stInitData.ModelParameters._R[9672] := 0.3081594558900842;
stInitData.ModelParameters._R[9673] := 0.49119037988082304;
stInitData.ModelParameters._R[9674] := 0.54802588103738414;
stInitData.ModelParameters._R[9675] := 0.5766695935703896;
stInitData.ModelParameters._R[9676] := 0.90517499100223242;
stInitData.ModelParameters._R[9677] := 0.32631200684456385;
stInitData.ModelParameters._R[9678] := 0.31554996521816614;
stInitData.ModelParameters._R[9679] := 0.58613432693044454;
stInitData.ModelParameters._R[9680] := 0.98725103325684738;
stInitData.ModelParameters._R[9681] := 0.39443656608666267;
stInitData.ModelParameters._R[9682] := 0.52590831780389014;
stInitData.ModelParameters._R[9683] := 0.33277164828551653;
stInitData.ModelParameters._R[9684] := 0.57697613821259108;
stInitData.ModelParameters._R[9685] := 0.59470626591824982;
stInitData.ModelParameters._R[9686] := 0.97728509593354573;
stInitData.ModelParameters._R[9687] := 0.6473974259604981;
stInitData.ModelParameters._R[9688] := 0.58921948813149061;
stInitData.ModelParameters._R[9689] := 0.77679355501374725;
stInitData.ModelParameters._R[9690] := 0.79979586848841022;
stInitData.ModelParameters._R[9691] := 0.20195251741029296;
stInitData.ModelParameters._R[9692] := 0.85091439584456219;
stInitData.ModelParameters._R[9693] := 0.27732676922075522;
stInitData.ModelParameters._R[9694] := 0.13292198388144139;
stInitData.ModelParameters._R[9695] := 0.27889231958345484;
stInitData.ModelParameters._R[9696] := 0.13763582277844255;
stInitData.ModelParameters._R[9697] := 0.33151232005878017;
stInitData.ModelParameters._R[9698] := 0.35145746439539727;
stInitData.ModelParameters._R[9699] := 0.36038726014308942;
stInitData.ModelParameters._R[9700] := 0.88193994244801943;
stInitData.ModelParameters._R[9701] := 0.9328112379804081;
stInitData.ModelParameters._R[9702] := 0.52121737425116754;
stInitData.ModelParameters._R[9703] := 0.7103941054557622;
stInitData.ModelParameters._R[9704] := 0.35591153481502213;
stInitData.ModelParameters._R[9705] := 0.30623573374135654;
stInitData.ModelParameters._R[9706] := 0.32448345869195733;
stInitData.ModelParameters._R[9707] := 0.25705792007434003;
stInitData.ModelParameters._R[9708] := 0.3001442867159051;
stInitData.ModelParameters._R[9709] := 0.71709970026557601;
stInitData.ModelParameters._R[9710] := 0.30537705430913215;
stInitData.ModelParameters._R[9711] := 0.40321743117402664;
stInitData.ModelParameters._R[9712] := 0.27289617464252264;
stInitData.ModelParameters._R[9713] := 0.57746419995378429;
stInitData.ModelParameters._R[9714] := 0.26762305834442551;
stInitData.ModelParameters._R[9715] := 0.2079714576941572;
stInitData.ModelParameters._R[9716] := 0.61443612128773306;
stInitData.ModelParameters._R[9717] := 0.14638196023715569;
stInitData.ModelParameters._R[9718] := 0.31171678328575386;
stInitData.ModelParameters._R[9719] := 0.17149049807118483;
stInitData.ModelParameters._R[9720] := 0.57987505218000635;
stInitData.ModelParameters._R[9721] := 0.59377132590735826;
stInitData.ModelParameters._R[9722] := 0.6228873515215011;
stInitData.ModelParameters._R[9723] := 0.35302883122952955;
stInitData.ModelParameters._R[9724] := 0.40866668302305986;
stInitData.ModelParameters._R[9725] := 0.39587181913887326;
stInitData.ModelParameters._R[9726] := 0.54428758424609014;
stInitData.ModelParameters._R[9727] := 0.74730280479554523;
stInitData.ModelParameters._R[9728] := 0.94126198539625039;
stInitData.ModelParameters._R[9729] := 0.75262284046442718;
stInitData.ModelParameters._R[9730] := 0.86419193265417726;
stInitData.ModelParameters._R[9731] := 0.97527451192212322;
stInitData.ModelParameters._R[9732] := 0.29691036623971701;
stInitData.ModelParameters._R[9733] := 0.3068750345184541;
stInitData.ModelParameters._R[9734] := 0.77801117617079574;
stInitData.ModelParameters._R[9735] := 0.52013899813102715;
stInitData.ModelParameters._R[9736] := 0.2159352389037883;
stInitData.ModelParameters._R[9737] := 0.48481560477638852;
stInitData.ModelParameters._R[9738] := 0.12702521089252394;
stInitData.ModelParameters._R[9739] := 0.23393696455088481;
stInitData.ModelParameters._R[9740] := 0.48627931050982687;
stInitData.ModelParameters._R[9741] := 0.78567517414504673;
stInitData.ModelParameters._R[9742] := 0.54289188771994268;
stInitData.ModelParameters._R[9743] := 0.35461820603697103;
stInitData.ModelParameters._R[9744] := 0.74780959726572205;
stInitData.ModelParameters._R[9745] := 0.67060317596121843;
stInitData.ModelParameters._R[9746] := 0.36062560169371338;
stInitData.ModelParameters._R[9747] := 0.76906602867914209;
stInitData.ModelParameters._R[9748] := 0.22247379637105591;
stInitData.ModelParameters._R[9749] := 0.96905625932380479;
stInitData.ModelParameters._R[9750] := 0.40699850966949458;
stInitData.ModelParameters._R[9751] := 0.79115939448714923;
stInitData.ModelParameters._R[9752] := 0.16890137358512397;
stInitData.ModelParameters._R[9753] := 0.42572836100797307;
stInitData.ModelParameters._R[9754] := 0.77986861062425639;
stInitData.ModelParameters._R[9755] := 0.96207793323773094;
stInitData.ModelParameters._R[9756] := 0.22836627769795068;
stInitData.ModelParameters._R[9757] := 0.36656334684361447;
stInitData.ModelParameters._R[9758] := 0.50011212685405437;
stInitData.ModelParameters._R[9759] := 0.10456968130595451;
stInitData.ModelParameters._R[9760] := 0.15291139386198394;
stInitData.ModelParameters._R[9761] := 0.72974999584542732;
stInitData.ModelParameters._R[9762] := 0.65151577378750392;
stInitData.ModelParameters._R[9763] := 0.72156165708286868;
stInitData.ModelParameters._R[9764] := 0.80533056043207263;
stInitData.ModelParameters._R[9765] := 0.3297540892709695;
stInitData.ModelParameters._R[9766] := 0.60249604863206108;
stInitData.ModelParameters._R[9767] := 0.29782552474488438;
stInitData.ModelParameters._R[9768] := 0.46509663904829945;
stInitData.ModelParameters._R[9769] := 0.83428493040856078;
stInitData.ModelParameters._R[9770] := 0.71249641952461906;
stInitData.ModelParameters._R[9771] := 0.30706070288783721;
stInitData.ModelParameters._R[9772] := 0.38961451708477912;
stInitData.ModelParameters._R[9773] := 0.28134385898356995;
stInitData.ModelParameters._R[9774] := 0.89810290091873457;
stInitData.ModelParameters._R[9775] := 0.62599877661269654;
stInitData.ModelParameters._R[9776] := 0.68892576012802009;
stInitData.ModelParameters._R[9777] := 0.35704014267279738;
stInitData.ModelParameters._R[9778] := 0.68552692558681905;
stInitData.ModelParameters._R[9779] := 0.46506801392177066;
stInitData.ModelParameters._R[9780] := 0.44827602984733361;
stInitData.ModelParameters._R[9781] := 0.60117405420418724;
stInitData.ModelParameters._R[9782] := 0.8598356559692204;
stInitData.ModelParameters._R[9783] := 0.14471334839153888;
stInitData.ModelParameters._R[9784] := 0.43374441264226504;
stInitData.ModelParameters._R[9785] := 0.83259316843209541;
stInitData.ModelParameters._R[9786] := 0.77691378154641844;
stInitData.ModelParameters._R[9787] := 0.41185978879895524;
stInitData.ModelParameters._R[9788] := 0.86809696188712371;
stInitData.ModelParameters._R[9789] := 0.45202449896875896;
stInitData.ModelParameters._R[9790] := 0.47387995480326295;
stInitData.ModelParameters._R[9791] := 0.37373938212944169;
stInitData.ModelParameters._R[9792] := 0.47203881799654901;
stInitData.ModelParameters._R[9793] := 0.21665736950560788;
stInitData.ModelParameters._R[9794] := 0.71193845643467191;
stInitData.ModelParameters._R[9795] := 0.60087178778721784;
stInitData.ModelParameters._R[9796] := 0.18480381185150935;
stInitData.ModelParameters._R[9797] := 0.61156038279243841;
stInitData.ModelParameters._R[9798] := 0.48881534640862712;
stInitData.ModelParameters._R[9799] := 0.2887492582190212;
stInitData.ModelParameters._R[9800] := 0.90560748438258731;
stInitData.ModelParameters._R[9801] := 0.91282438528684806;
stInitData.ModelParameters._R[9802] := 0.93933814790319115;
stInitData.ModelParameters._R[9803] := 0.46333753107322218;
stInitData.ModelParameters._R[9804] := 0.50569000162206179;
stInitData.ModelParameters._R[9805] := 0.30566404573220807;
stInitData.ModelParameters._R[9806] := 0.64965225594956377;
stInitData.ModelParameters._R[9807] := 0.70292342688034215;
stInitData.ModelParameters._R[9808] := 0.13905092695678048;
stInitData.ModelParameters._R[9809] := 0.97994981053390018;
stInitData.ModelParameters._R[9810] := 0.43445130700397561;
stInitData.ModelParameters._R[9811] := 0.31506443138868001;
stInitData.ModelParameters._R[9812] := 0.85757506749587809;
stInitData.ModelParameters._R[9813] := 0.1763294640582358;
stInitData.ModelParameters._R[9814] := 0.69769559239292012;
stInitData.ModelParameters._R[9815] := 0.98351187446968924;
stInitData.ModelParameters._R[9816] := 0.98809332311749754;
stInitData.ModelParameters._R[9817] := 0.24972506295303096;
stInitData.ModelParameters._R[9818] := 0.29677807389335964;
stInitData.ModelParameters._R[9819] := 0.7310455966023609;
stInitData.ModelParameters._R[9820] := 0.70509892202199953;
stInitData.ModelParameters._R[9821] := 0.86081634813716212;
stInitData.ModelParameters._R[9822] := 0.18440328527322083;
stInitData.ModelParameters._R[9823] := 0.79295740209692889;
stInitData.ModelParameters._R[9824] := 0.21655927614605064;
stInitData.ModelParameters._R[9825] := 0.81458404577631305;
stInitData.ModelParameters._R[9826] := 0.91417569866210047;
stInitData.ModelParameters._R[9827] := 0.53598273335743885;
stInitData.ModelParameters._R[9828] := 0.13001393050244439;
stInitData.ModelParameters._R[9829] := 0.42674438764497558;
stInitData.ModelParameters._R[9830] := 0.43386560348008019;
stInitData.ModelParameters._R[9831] := 0.92167093241993181;
stInitData.ModelParameters._R[9832] := 0.53657613107005286;
stInitData.ModelParameters._R[9833] := 0.47039575501314101;
stInitData.ModelParameters._R[9834] := 0.12185679425336628;
stInitData.ModelParameters._R[9835] := 0.69983295137423684;
stInitData.ModelParameters._R[9836] := 0.33035427524428851;
stInitData.ModelParameters._R[9837] := 0.95589594052270166;
stInitData.ModelParameters._R[9838] := 0.88544502057114216;
stInitData.ModelParameters._R[9839] := 0.21414976605871799;
stInitData.ModelParameters._R[9840] := 0.3238939102341406;
stInitData.ModelParameters._R[9841] := 0.77378392527788453;
stInitData.ModelParameters._R[9842] := 0.96786698139501082;
stInitData.ModelParameters._R[9843] := 0.11756317333129397;
stInitData.ModelParameters._R[9844] := 0.81129960834296344;
stInitData.ModelParameters._R[9845] := 0.11523464413150972;
stInitData.ModelParameters._R[9846] := 0.21190597514665205;
stInitData.ModelParameters._R[9847] := 0.25786608897761082;
stInitData.ModelParameters._R[9848] := 0.58976475816634866;
stInitData.ModelParameters._R[9849] := 0.18870306172612777;
stInitData.ModelParameters._R[9850] := 0.24374627352027151;
stInitData.ModelParameters._R[9851] := 0.59687413219332952;
stInitData.ModelParameters._R[9852] := 0.88938063303810577;
stInitData.ModelParameters._R[9853] := 0.48799895426478723;
stInitData.ModelParameters._R[9854] := 0.66841219131362539;
stInitData.ModelParameters._R[9855] := 0.36963265944559598;
stInitData.ModelParameters._R[9856] := 0.82943424578666913;
stInitData.ModelParameters._R[9857] := 0.52837834484509139;
stInitData.ModelParameters._R[9858] := 0.78124555273882812;
stInitData.ModelParameters._R[9859] := 0.89411646635390996;
stInitData.ModelParameters._R[9860] := 0.44655796563814998;
stInitData.ModelParameters._R[9861] := 0.26907291506530817;
stInitData.ModelParameters._R[9862] := 0.90306949756615351;
stInitData.ModelParameters._R[9863] := 0.49719892918312592;
stInitData.ModelParameters._R[9864] := 0.39060635402980037;
stInitData.ModelParameters._R[9865] := 0.56296943485308804;
stInitData.ModelParameters._R[9866] := 0.60029370508560109;
stInitData.ModelParameters._R[9867] := 0.20633785991571885;
stInitData.ModelParameters._R[9868] := 0.75394922437920553;
stInitData.ModelParameters._R[9869] := 0.51501421427446903;
stInitData.ModelParameters._R[9870] := 0.6656375285467182;
stInitData.ModelParameters._R[9871] := 0.8977548300710646;
stInitData.ModelParameters._R[9872] := 0.68278844051304932;
stInitData.ModelParameters._R[9873] := 0.61816206649149363;
stInitData.ModelParameters._R[9874] := 0.91143009974599742;
stInitData.ModelParameters._R[9875] := 0.94326207364445436;
stInitData.ModelParameters._R[9876] := 0.5115350512905229;
stInitData.ModelParameters._R[9877] := 0.24682020951989475;
stInitData.ModelParameters._R[9878] := 0.18152125255983564;
stInitData.ModelParameters._R[9879] := 0.77840909392712043;
stInitData.ModelParameters._R[9880] := 0.383904375066493;
stInitData.ModelParameters._R[9881] := 0.21915716447704253;
stInitData.ModelParameters._R[9882] := 0.56995532127121473;
stInitData.ModelParameters._R[9883] := 0.40433296362694537;
stInitData.ModelParameters._R[9884] := 0.11836991444730471;
stInitData.ModelParameters._R[9885] := 0.90923916899573165;
stInitData.ModelParameters._R[9886] := 0.58802008711548659;
stInitData.ModelParameters._R[9887] := 0.75842061053208376;
stInitData.ModelParameters._R[9888] := 0.65446898207421211;
stInitData.ModelParameters._R[9889] := 0.32221721211912274;
stInitData.ModelParameters._R[9890] := 0.48455431451698294;
stInitData.ModelParameters._R[9891] := 0.22037638529936665;
stInitData.ModelParameters._R[9892] := 0.24955994595845665;
stInitData.ModelParameters._R[9893] := 0.6046791376096643;
stInitData.ModelParameters._R[9894] := 0.34097230707455695;
stInitData.ModelParameters._R[9895] := 0.26855284583115951;
stInitData.ModelParameters._R[9896] := 0.82031413680043519;
stInitData.ModelParameters._R[9897] := 0.89125135895419438;
stInitData.ModelParameters._R[9898] := 0.76446758389946656;
stInitData.ModelParameters._R[9899] := 0.52695820601449106;
stInitData.ModelParameters._R[9900] := 0.27559007504240551;
stInitData.ModelParameters._R[9901] := 0.10212010932597458;
stInitData.ModelParameters._R[9902] := 0.1242068193691995;
stInitData.ModelParameters._R[9903] := 0.37788681109071742;
stInitData.ModelParameters._R[9904] := 0.83272941043909587;
stInitData.ModelParameters._R[9905] := 0.26340634971484178;
stInitData.ModelParameters._R[9906] := 0.18218572649490977;
stInitData.ModelParameters._R[9907] := 0.32245904283530485;
stInitData.ModelParameters._R[9908] := 0.86568668088888945;
stInitData.ModelParameters._R[9909] := 0.13974802192888491;
stInitData.ModelParameters._R[9910] := 0.59516193834479858;
stInitData.ModelParameters._R[9911] := 0.76483707879202056;
stInitData.ModelParameters._R[9912] := 0.51143841182357086;
stInitData.ModelParameters._R[9913] := 0.39162845679447655;
stInitData.ModelParameters._R[9914] := 0.53876455011802438;
stInitData.ModelParameters._R[9915] := 0.45695097931081197;
stInitData.ModelParameters._R[9916] := 0.24462842999048356;
stInitData.ModelParameters._R[9917] := 0.53046316360152046;
stInitData.ModelParameters._R[9918] := 0.54925684421213938;
stInitData.ModelParameters._R[9919] := 0.51839003720238519;
stInitData.ModelParameters._R[9920] := 0.97064456541005695;
stInitData.ModelParameters._R[9921] := 0.5085792426367588;
stInitData.ModelParameters._R[9922] := 0.25989320732517956;
stInitData.ModelParameters._R[9923] := 0.67273895419636554;
stInitData.ModelParameters._R[9924] := 0.43178574153741212;
stInitData.ModelParameters._R[9925] := 0.67761621816188444;
stInitData.ModelParameters._R[9926] := 0.89537055173038982;
stInitData.ModelParameters._R[9927] := 0.37394490472178032;
stInitData.ModelParameters._R[9928] := 0.42633607011448826;
stInitData.ModelParameters._R[9929] := 0.95461521398069504;
stInitData.ModelParameters._R[9930] := 0.12157880126117859;
stInitData.ModelParameters._R[9931] := 0.34322859860874877;
stInitData.ModelParameters._R[9932] := 0.67040877835156609;
stInitData.ModelParameters._R[9933] := 0.50805909243936709;
stInitData.ModelParameters._R[9934] := 0.33646038691757413;
stInitData.ModelParameters._R[9935] := 0.50487648159022047;
stInitData.ModelParameters._R[9936] := 0.48474990849157351;
stInitData.ModelParameters._R[9937] := 0.83218824319015583;
stInitData.ModelParameters._R[9938] := 0.58104809770634869;
stInitData.ModelParameters._R[9939] := 0.99475295605039737;
stInitData.ModelParameters._R[9940] := 0.96769216848124218;
stInitData.ModelParameters._R[9941] := 0.98801487477731365;
stInitData.ModelParameters._R[9942] := 0.60904945047017345;
stInitData.ModelParameters._R[9943] := 0.2646022736436987;
stInitData.ModelParameters._R[9944] := 0.7414170990710871;
stInitData.ModelParameters._R[9945] := 0.731903915379436;
stInitData.ModelParameters._R[9946] := 0.32519407164893999;
stInitData.ModelParameters._R[9947] := 0.87587235810615294;
stInitData.ModelParameters._R[9948] := 0.19665848717129264;
stInitData.ModelParameters._R[9949] := 0.10971892485465168;
stInitData.ModelParameters._R[9950] := 0.50439342672529575;
stInitData.ModelParameters._R[9951] := 0.22104375737750892;
stInitData.ModelParameters._R[9952] := 0.70265879009455434;
stInitData.ModelParameters._R[9953] := 0.95769300417984582;
stInitData.ModelParameters._R[9954] := 0.90474959849072878;
stInitData.ModelParameters._R[9955] := 0.68454510827887072;
stInitData.ModelParameters._R[9956] := 0.37560133540865548;
stInitData.ModelParameters._R[9957] := 0.77528505338122833;
stInitData.ModelParameters._R[9958] := 0.89090794989770672;
stInitData.ModelParameters._R[9959] := 0.33569319079658316;
stInitData.ModelParameters._R[9960] := 0.57809660926134632;
stInitData.ModelParameters._R[9961] := 0.44644731935988691;
stInitData.ModelParameters._R[9962] := 0.66518006373582306;
stInitData.ModelParameters._R[9963] := 0.11587791613012297;
stInitData.ModelParameters._R[9964] := 0.66962135407134016;
stInitData.ModelParameters._R[9965] := 0.65411366157139339;
stInitData.ModelParameters._R[9966] := 0.17122153339532498;
stInitData.ModelParameters._R[9967] := 0.65456614211153696;
stInitData.ModelParameters._R[9968] := 0.43822114656284816;
stInitData.ModelParameters._R[9969] := 0.99167526978973231;
stInitData.ModelParameters._R[9970] := 0.17130083757899073;
stInitData.ModelParameters._R[9971] := 0.80896981999928896;
stInitData.ModelParameters._R[9972] := 0.1392228323239931;
stInitData.ModelParameters._R[9973] := 0.26002489094372727;
stInitData.ModelParameters._R[9974] := 0.29932156047613284;
stInitData.ModelParameters._R[9975] := 0.44787972455385927;
stInitData.ModelParameters._R[9976] := 0.15553405240966153;
stInitData.ModelParameters._R[9977] := 0.23350331154732545;
stInitData.ModelParameters._R[9978] := 0.47331829827625882;
stInitData.ModelParameters._R[9979] := 0.3882417694413709;
stInitData.ModelParameters._R[9980] := 0.92125079992584169;
stInitData.ModelParameters._R[9981] := 0.40443966574410983;
stInitData.ModelParameters._R[9982] := 0.48363194330410331;
stInitData.ModelParameters._R[9983] := 0.26192827347621206;
stInitData.ModelParameters._R[9984] := 0.7233345632922894;
stInitData.ModelParameters._R[9985] := 0.86198415078593116;
stInitData.ModelParameters._R[9986] := 0.30317141165406225;
stInitData.ModelParameters._R[9987] := 0.80736452653961532;
stInitData.ModelParameters._R[9988] := 0.21411526103256506;
stInitData.ModelParameters._R[9989] := 0.92136268137212762;
stInitData.ModelParameters._R[9990] := 0.85098137072645996;
stInitData.ModelParameters._R[9991] := 0.38588205697320843;
stInitData.ModelParameters._R[9992] := 0.94033745731254381;
stInitData.ModelParameters._R[9993] := 0.61159251874644449;
stInitData.ModelParameters._R[9994] := 0.98794924687276686;
stInitData.ModelParameters._R[9995] := 0.35299145227964646;
stInitData.ModelParameters._R[9996] := 0.15472474018185081;
stInitData.ModelParameters._R[9997] := 0.70343753151491384;
stInitData.ModelParameters._R[9998] := 0.55134249842269067;
stInitData.ModelParameters._R[9999] := 0.27327354697297446;
stInitData.ModelParameters.WS_MAX_LENGTHS := -0.10000000000000001;
stInitData.ModelParameters.WS_MAX_VEL_m_s := 0.40000000000000002;
stInitData.ModelParameters.WS_MIN_LENGTHS := -0.20000000000000001;
stInitData.ModelParameters.duration := 1;
stInitData.ModelParameters.zero_poses := 3143153400;
stInitData.ModelParameters.CompareToConstant1_const := 0.5;
stInitData.ModelParameters.CompareToConstant2_const := 4.5;
stInitData.ModelParameters.DetectChange_vinit := 0;
stInitData.ModelParameters.RESETconst_Value := 0;
stInitData.ModelParameters.Constant4_Value := 3;
stInitData.ModelParameters.w_Y0 := 0;
stInitData.ModelParameters.delay_counter_Y0 := 0;
stInitData.ModelParameters.Constant_Value := 1;
stInitData.ModelParameters.Constant1_Value := 2;
stInitData.ModelParameters.Integrator_IC := 0;
stInitData.ModelParameters.TransferFcn_A[0] := -20;
stInitData.ModelParameters.TransferFcn_A[1] := -99.999999999999986;
stInitData.ModelParameters.TransferFcn_C[0] := 0;
stInitData.ModelParameters.TransferFcn_C[1] := 99.999999999999986;
stInitData.ModelParameters.Switch_Threshold := -1;
stInitData.ModelParameters.Out1_Y0 := 0;
stInitData.ModelParameters.Constant_Value_g := 0;
stInitData.ModelParameters.UnitDelay_InitialCondition := 0;
stInitData.ModelParameters.FixPtConstant_Value := 1;
stInitData.ModelParameters.BREAKFLAG_Value := 1;
stInitData.ModelParameters.Saturation1_UpperSat := 1;
stInitData.ModelParameters.Saturation1_LowerSat := 0;
stInitData.ModelParameters.velBREAK_FLAG_Value := 1;
stInitData.ModelParameters.Constant1_Value_b := -1;
stInitData.ModelParameters.Memory_InitialCondition := 0;
stInitData.ModelParameters.Saturation3_UpperSat := 1.7976931348623157e+308;
stInitData.ModelParameters.Saturation3_LowerSat := 0;
stInitData.ModelParameters.lenBREAK_FLAG_Value := 1;
stInitData.ModelParameters.Constant1_Value_d := -1;
stInitData.ModelParameters.Gain1_Gain := -1;
stInitData.ModelParameters.Saturation4_UpperSat := 1.7976931348623157e+308;
stInitData.ModelParameters.Saturation4_LowerSat := 0;
stInitData.ModelParameters.colBREAK_FLAG_Value := 0;
stInitData.ModelParameters.Constant1_Value_a := -1;
stInitData.ModelParameters.Constant1_Value_k := 600;
stInitData.ModelParameters.TorqueGAIN_Gain := 1;
stInitData.ModelParameters.m_endeff_Value := 0.14499999999999999;
stInitData.ModelParameters.delays_Value := 0.01;
stInitData.ModelParameters.Memory_InitialCondition_a := 0;
stInitData.ModelParameters.Saturation5_UpperSat := 1.7976931348623157e+308;
stInitData.ModelParameters.Saturation5_LowerSat := 0;
stInitData.ModelParameters.Saturation_UpperSat := 1;
stInitData.ModelParameters.Saturation_LowerSat := 0;
stInitData.ModelParameters.Gain_Gain := 200;
stInitData.ModelParameters.BreakValue_UpperSat := 1;
stInitData.ModelParameters.BreakValue_LowerSat := 0;
stInitData.ModelParameters.BREAKconst_Value := 6;
stInitData.ModelParameters.INITconst_Value := 0;
stInitData.ModelParameters.Delay_InitialCondition := 0;
stInitData.ModelParameters.Constant3_Value := 1;
stInitData.ModelParameters.Constant_Value_k := 1;
stInitData.ModelParameters.Integrator_IC_n := 0;
stInitData.ModelParameters.Delay_InitialCondition_l := 0;
stInitData.ModelParameters.Constant6_Value := 1;
stInitData.ModelParameters.Constant9_Value := 0;
stInitData.ModelParameters.Integrator1_IC := 0;
stInitData.ModelParameters.SineWave_Amp := 0.5;
stInitData.ModelParameters.SineWave_Bias := 0.5;
stInitData.ModelParameters.SineWave_Freq := 0.10000000000000001;
stInitData.ModelParameters.SineWave_Phase := 0;
stInitData.ModelParameters.Constant12_Value := 0;
stInitData.ModelParameters.Integrator1_IC_b := 0;
stInitData.ModelParameters.TransferFcn1_A[0] := -200;
stInitData.ModelParameters.TransferFcn1_A[1] := -10000;
stInitData.ModelParameters.TransferFcn1_C[0] := 0;
stInitData.ModelParameters.TransferFcn1_C[1] := 10000;
stInitData.ModelParameters.TransferFcn2_A[0] := -20;
stInitData.ModelParameters.TransferFcn2_A[1] := -100;
stInitData.ModelParameters.TransferFcn2_C[0] := 0;
stInitData.ModelParameters.TransferFcn2_C[1] := 100;
stInitData.ModelParameters.Constant2_Value := -2;
stInitData.ModelParameters.Integrator_IC_k := 0;
stInitData.ModelParameters.Saturation_UpperSat_c := 1;
stInitData.ModelParameters.Saturation_LowerSat_b := 0.10000000000000001;
stInitData.ModelParameters.select_w_Value := 1;
stInitData.ModelParameters.VorsteuerungfrMotorkraftohneRei := 2;
stInitData.ModelParameters.Constant7_Value := 1;
stInitData.ModelParameters.torque_scaling_Value := 250;
stInitData.ModelParameters.enableBrakeTorque_FLAG_Value := 1;
stInitData.ModelParameters.UnitDelay_InitialCondition_g[0] := 0;
stInitData.ModelParameters.UnitDelay_InitialCondition_g[1] := 0;
stInitData.ModelParameters.UnitDelay_InitialCondition_g[2] := 0;
stInitData.ModelParameters.UnitDelay_InitialCondition_g[3] := 0;
stInitData.ModelParameters.UnitDelay_InitialCondition_g[4] := 0;
stInitData.ModelParameters.UnitDelay_InitialCondition_g[5] := 0;
stInitData.ModelParameters.UnitDelay_InitialCondition_g[6] := 0;
stInitData.ModelParameters.UnitDelay_InitialCondition_g[7] := 0;
stInitData.ModelParameters.UnitDelay_InitialCondition_g[8] := 0;
stInitData.ModelParameters.UnitDelay_InitialCondition_g[9] := 0;
stInitData.ModelParameters.UnitDelay_InitialCondition_g[10] := 0;
stInitData.ModelParameters.UnitDelay_InitialCondition_g[11] := 0;
stInitData.ModelParameters.UnitDelay_InitialCondition_g[12] := 0;
stInitData.ModelParameters.UnitDelay_InitialCondition_g[13] := 0;
stInitData.ModelParameters.UnitDelay_InitialCondition_g[14] := 0;
stInitData.ModelParameters.UnitDelay_InitialCondition_g[15] := 0;
stInitData.ModelParameters.UnitDelay_InitialCondition_g[16] := 0;
stInitData.ModelParameters.UnitDelay_InitialCondition_g[17] := 0;
stInitData.ModelParameters.UnitDelay_InitialCondition_g[18] := 0;
stInitData.ModelParameters.UnitDelay_InitialCondition_g[19] := 0;
stInitData.ModelParameters.UnitDelay_InitialCondition_l[0] := 0;
stInitData.ModelParameters.UnitDelay_InitialCondition_l[1] := 0;
stInitData.ModelParameters.UnitDelay_InitialCondition_l[2] := 0;
stInitData.ModelParameters.UnitDelay_InitialCondition_l[3] := 0;
stInitData.ModelParameters.UnitDelay_InitialCondition_l[4] := 0;
stInitData.ModelParameters.UnitDelay_InitialCondition_l[5] := 0;
stInitData.ModelParameters.UnitDelay_InitialCondition_l[6] := 0;
stInitData.ModelParameters.UnitDelay_InitialCondition_l[7] := 0;
stInitData.ModelParameters.UnitDelay_InitialCondition_l[8] := 0;
stInitData.ModelParameters.UnitDelay_InitialCondition_l[9] := 0;
stInitData.ModelParameters.UnitDelay_InitialCondition_l[10] := 0;
stInitData.ModelParameters.UnitDelay_InitialCondition_l[11] := 0;
stInitData.ModelParameters.UnitDelay_InitialCondition_l[12] := 0;
stInitData.ModelParameters.UnitDelay_InitialCondition_l[13] := 0;
stInitData.ModelParameters.UnitDelay_InitialCondition_l[14] := 0;
stInitData.ModelParameters.UnitDelay_InitialCondition_l[15] := 0;
stInitData.ModelParameters.UnitDelay_InitialCondition_l[16] := 0;
stInitData.ModelParameters.UnitDelay_InitialCondition_l[17] := 0;
stInitData.ModelParameters.UnitDelay_InitialCondition_l[18] := 0;
stInitData.ModelParameters.UnitDelay_InitialCondition_l[19] := 0;
stInitData.ModelParameters.Constant5_Value := -1;
stInitData.ModelParameters.UnitDelay_InitialCondition_o[0] := 0;
stInitData.ModelParameters.UnitDelay_InitialCondition_o[1] := 0;
stInitData.ModelParameters.UnitDelay_InitialCondition_o[2] := 0;
stInitData.ModelParameters.UnitDelay_InitialCondition_o[3] := 0;
stInitData.ModelParameters.UnitDelay_InitialCondition_o[4] := 0;
stInitData.ModelParameters.UnitDelay_InitialCondition_o[5] := 0;
stInitData.ModelParameters.UnitDelay_InitialCondition_o[6] := 0;
stInitData.ModelParameters.UnitDelay_InitialCondition_o[7] := 0;
stInitData.ModelParameters.UnitDelay_InitialCondition_o[8] := 0;
stInitData.ModelParameters.UnitDelay_InitialCondition_o[9] := 0;
stInitData.ModelParameters.UnitDelay_InitialCondition_o[10] := 0;
stInitData.ModelParameters.UnitDelay_InitialCondition_o[11] := 0;
stInitData.ModelParameters.UnitDelay_InitialCondition_o[12] := 0;
stInitData.ModelParameters.UnitDelay_InitialCondition_o[13] := 0;
stInitData.ModelParameters.UnitDelay_InitialCondition_o[14] := 0;
stInitData.ModelParameters.UnitDelay_InitialCondition_o[15] := 0;
stInitData.ModelParameters.UnitDelay_InitialCondition_o[16] := 0;
stInitData.ModelParameters.UnitDelay_InitialCondition_o[17] := 0;
stInitData.ModelParameters.UnitDelay_InitialCondition_o[18] := 0;
stInitData.ModelParameters.UnitDelay_InitialCondition_o[19] := 0;
stInitData.ModelParameters.dms_offset_Value := -202000;
stInitData.ModelParameters.Gain1_Gain_f := 5.6690000000000003e-07;
stInitData.ModelParameters.UnitDelay_InitialCondition_j[0] := 0;
stInitData.ModelParameters.UnitDelay_InitialCondition_j[1] := 0;
stInitData.ModelParameters.UnitDelay_InitialCondition_j[2] := 0;
stInitData.ModelParameters.UnitDelay_InitialCondition_j[3] := 0;
stInitData.ModelParameters.UnitDelay_InitialCondition_j[4] := 0;
stInitData.ModelParameters.UnitDelay_InitialCondition_j[5] := 0;
stInitData.ModelParameters.UnitDelay_InitialCondition_j[6] := 0;
stInitData.ModelParameters.UnitDelay_InitialCondition_j[7] := 0;
stInitData.ModelParameters.UnitDelay_InitialCondition_j[8] := 0;
stInitData.ModelParameters.UnitDelay_InitialCondition_j[9] := 0;
stInitData.ModelParameters.UnitDelay_InitialCondition_j[10] := 0;
stInitData.ModelParameters.UnitDelay_InitialCondition_j[11] := 0;
stInitData.ModelParameters.UnitDelay_InitialCondition_j[12] := 0;
stInitData.ModelParameters.UnitDelay_InitialCondition_j[13] := 0;
stInitData.ModelParameters.UnitDelay_InitialCondition_j[14] := 0;
stInitData.ModelParameters.UnitDelay_InitialCondition_j[15] := 0;
stInitData.ModelParameters.UnitDelay_InitialCondition_j[16] := 0;
stInitData.ModelParameters.UnitDelay_InitialCondition_j[17] := 0;
stInitData.ModelParameters.UnitDelay_InitialCondition_j[18] := 0;
stInitData.ModelParameters.UnitDelay_InitialCondition_j[19] := 0;
stInitData.ModelParameters.Constant10_Value := 0;
stInitData.ModelParameters.Constant2_Value_b := 1;
stInitData.ModelParameters.Constant_Value_d := 1;
stInitData.ModelParameters.Delay_DelayLength := 10000;
stInitData.ModelParameters.Delay_DelayLength_a := 1;
stInitData.ModelParameters.RESET_CurrentSetting := 0;
stInitData.ContextInfoArr_0_TaskOidHdr.indexGroup := 0;
stInitData.ContextInfoArr_0_TaskOidHdr.indexOffset := 16#03002060;
stInitData.ContextInfoArr_0_TaskOidHdr.cbData := SIZEOF(stInitData.ContextInfoArr_0_TaskOid);
stInitData.ContextInfoArr_0_TaskPriorityHdr.indexGroup := 0;
stInitData.ContextInfoArr_0_TaskPriorityHdr.indexOffset := 16#03002070;
stInitData.ContextInfoArr_0_TaskPriorityHdr.cbData := SIZEOF(stInitData.ContextInfoArr_0_TaskPriority);
stInitData.ContextInfoArr_0_TaskCycleTimeNsHdr.indexGroup := 0;
stInitData.ContextInfoArr_0_TaskCycleTimeNsHdr.indexOffset := 16#03002080;
stInitData.ContextInfoArr_0_TaskCycleTimeNsHdr.cbData := SIZEOF(stInitData.ContextInfoArr_0_TaskCycleTimeNs);
stInitData.ContextInfoArr_0_TaskPortHdr.indexGroup := 0;
stInitData.ContextInfoArr_0_TaskPortHdr.indexOffset := 16#03002090;
stInitData.ContextInfoArr_0_TaskPortHdr.cbData := SIZEOF(stInitData.ContextInfoArr_0_TaskPort);
stInitData.ContextInfoArr_0_TaskSortOrderHdr.indexGroup := 0;
stInitData.ContextInfoArr_0_TaskSortOrderHdr.indexOffset := 16#030020b0;
stInitData.ContextInfoArr_0_TaskSortOrderHdr.cbData := SIZEOF(stInitData.ContextInfoArr_0_TaskSortOrder);
stInitData.Header.cbData := SIZEOF(stInitData)-SIZEOF(stInitData.Header);
stInitData.Header.uiElmCnt := 11;


// set pointer to InitData structure
SetInitDataInfo(ADR(stInitData));

// set DataArea information
SetDataAreaInfo(ADR(arrDataAreas),2);
arrDataAreas[1].nDataAreaId := 0;
arrDataAreas[1].nSize := SIZEOF(stInput);
arrDataAreas[1].pPlcVar := ADR(stInput);
arrDataAreas[1].pModuleProcImg := 0;
arrDataAreas[1].eDataAreaType := E_TcMatSimDataAreaType.InputDst;
arrDataAreas[2].nDataAreaId := 1;
arrDataAreas[2].nSize := SIZEOF(stOutput);
arrDataAreas[2].pPlcVar := ADR(stOutput);
arrDataAreas[2].pModuleProcImg := 0;
arrDataAreas[2].eDataAreaType := E_TcMatSimDataAreaType.OutputSrc;


// initialize basic interface pointers and return
FB_init := SUCCEEDED(Init(oid));
                  
                
END_METHOD

METHOD Execute : HRESULT
                  
IF (SUCCEEDED(hResult)) THEN
  hResult := VerifyParameters();
END_IF

// update DataArea information
SetDataAreaInfo(ADR(arrDataAreas),2);
arrDataAreas[1].nDataAreaId := 0;
arrDataAreas[1].nSize := SIZEOF(stInput);
arrDataAreas[1].pPlcVar := ADR(stInput);
arrDataAreas[1].pModuleProcImg := 0;
arrDataAreas[1].eDataAreaType := E_TcMatSimDataAreaType.InputDst;
arrDataAreas[2].nDataAreaId := 1;
arrDataAreas[2].nSize := SIZEOF(stOutput);
arrDataAreas[2].pPlcVar := ADR(stOutput);
arrDataAreas[2].pModuleProcImg := 0;
arrDataAreas[2].eDataAreaType := E_TcMatSimDataAreaType.OutputSrc;

	
// call base method
Execute := SUPER^.Execute();
                  
                
END_METHOD

{attribute 'object_name' := 'VerifyParameters'}
METHOD VerifyParameters : HRESULT
  VAR
    moduleCallByParam : TctModuleCallByType;
  END_VAR
                  
IF (bParametersVerified) THEN
  VerifyParameters := Tc2_System.E_HRESULTAdsErr.HRESULT_ADS_NOERROR;
ELSE
  VerifyParameters := GetObjPara(stInitData.CallByHdr.indexOffset,SIZEOF(moduleCallByParam),ADR(moduleCallByParam));
  
  // check the "CallBy" parameter to be set to "Module"
  IF (SUCCEEDED(VerifyParameters) AND (moduleCallByParam <> TctModuleCallByType.Module)) THEN
      VerifyParameters := Tc2_System.E_HRESULTAdsErr.INVALIDPARM;
  END_IF
  
  // set the parameters verified flag
  bParametersVerified := SUCCEEDED(VerifyParameters);
END_IF
                  
                
END_METHOD

PROPERTY InitData : ST_RL_Learn_DirectControlInitData
GET
                    InitData := stInitData;
                  
END_GET
SET
                    stInitData := InitData;
                  
END_SET
END_PROPERTY
END_FUNCTION_BLOCK
